(* CoDeSys 2.3.9.41 project: testUPC.pro *)
(* Libraries: Standard.lib 4.10.05 11:14:46, IecSfc.lib 13.4.06 15:51:28, SYSLIBCALLBACK.LIB 26.9.08 16:43:52 *)

(* POU PLC_PRG, ST *)
PROGRAM PLC_PRG
VAR
	RS1: RS;
END_VAR
VAR_OUTPUT
	DO_xEmitter: BOOL;
	DO_xRemover: BOOL;
	DO_xStartLedButton: BOOL;
	DO_xStopLedButton: BOOL;
	DO_xStartLed: BOOL;
	DO_xStopLed: BOOL;
	DO_xConveerOne: BOOL;
	DO_xAlarmLed: BOOL;
	DO_xAlarmZoom: BOOL;
	AO_wConveerTwo: USINT;
END_VAR
VAR_INPUT
	DI_xStart: BOOL;
	DI_xStop: BOOL;
	DI_xAlarmStop: BOOL;
	AI_wPotentiommetr: USINT;

END_VAR
(*Инициализация эмиттеров и ремуверов*)
DO_xEmitter:=DO_xRemover:=TRUE;

(*запуск конвееров и кнопки управления*)
RS1(SET := DI_xStart, RESET1 := NOT DI_xStop OR NOT DI_xAlarmStop);
DO_xStartLedButton := (DI_xStart);
DO_xStopLedButton := (NOT DI_xStop);
DO_xConveerOne := DO_xStartLed := RS1.Q1;
IF(RS1.Q1 AND AI_wPotentiommetr > 5) THEN
	AO_wConveerTwo := AI_wPotentiommetr;
ELSIF(RS1.Q1 AND AI_wPotentiommetr<=5) THEN
	AO_wConveerTwo := 5;
ELSE
	AO_wConveerTwo := 0;
END_IF;
DO_xStopLed := NOT RS1.Q1;
DO_xAlarmLed := DO_xAlarmZoom := NOT DI_xAlarmStop;
END_PROGRAM
